// TIA Portal V16 export
// export: Created 2021-09-08T12:44:31.9643726Z, ExportSetting WithDefaults, DisplayName Totally Integrated Automation Portal, DisplayVersion V16 Update 3, DisplayName TIA Portal Version Control Interface, DisplayVersion V16 Update 2, DisplayName TIA Portal Openness, DisplayVersion V16 Update 3, DisplayName TIA Portal Teamcenter Gateway, DisplayVersion V16, DisplayName STEP 7 Professional, DisplayVersion V16 Update 3, DisplayName STEP 7 Safety, DisplayVersion V16, DisplayName WinCC Advanced, DisplayVersion V16 Update 3
VAR_GLOBAL   // PLC tag table "A1_AQ"
   AO_DVA503_Setting AT %QW64 : Int;   // DVA503 Стан
   AO_DVA510_Setting AT %QW66 : Int;   // DVA510 Стан
END_VAR
VAR_GLOBAL CONSTANT   // user constants
   "qwDVA-503_Setting" : Int := 0;
   "qw_DVA-510_Setting" : Int := 1;
END_VAR
